FUNCTION_BLOCK Multicast_Client (* Basic Function Block Type *)
  (* Standard: 61499-2 *)
  (* Version 0.2, 2003-12-04, JHC, Rockwell Automation, Renamed for better indexing. *)
  (* Version 0.1, 2002-11-05, JHC, Rockwell Automation, Corrected missing ST element in Algorithm REQ. *)
  (* Version 0.0, 2000-05-30, JHC, Rockwell Automation *)
  (* Compiler header: package fb.rt.cs725; *)
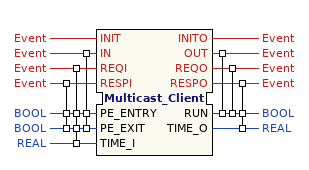
  EVENT_INPUT
    INIT; (* Initialization Request *)
    IN WITH PE_ENTRY, PE_EXIT;
    REQI WITH PE_ENTRY, PE_EXIT, TIME_I;
    RESPI WITH PE_ENTRY, PE_EXIT;
  END_EVENT
  EVENT_OUTPUT
    INITO; (* Initialization Confirm *)
    OUT WITH RUN;
    REQO WITH RUN;
    RESPO WITH RUN, TIME_O;
  END_EVENT
  VAR_INPUT
    PE_ENTRY : BOOL;
    PE_EXIT : BOOL;
    TIME_I : REAL;
  END_VAR
  VAR_OUTPUT
    RUN : BOOL;
    TIME_O : REAL;
  END_VAR
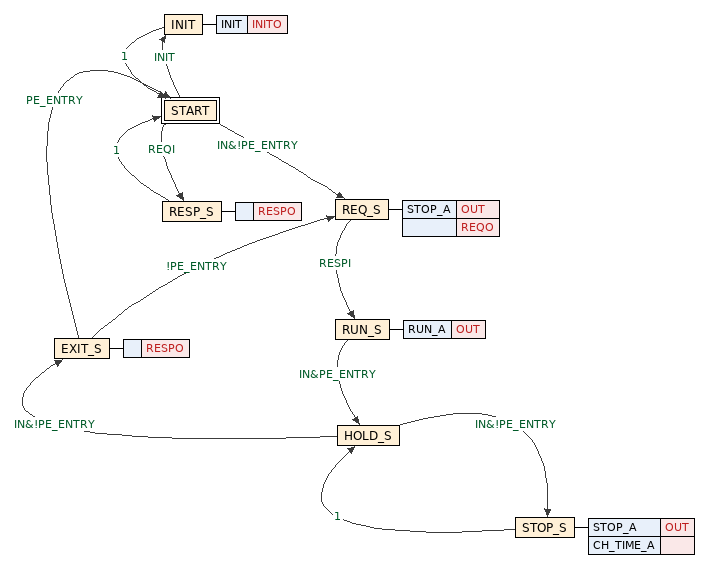
  EC_STATES
    START; (* Initial State *)
    INIT : INIT -> INITO; (* Initialization *)
    REQ_S : STOP_A -> OUT, -> REQO;
    RUN_S : RUN_A -> OUT;
    RESP_S : -> RESPO;
    EXIT_S : -> RESPO;
    STOP_S : STOP_A -> OUT, CH_TIME_A;
    HOLD_S;
  END_STATES
  EC_TRANSITIONS
    START TO INIT := INIT;
    INIT TO START := 1;
    START TO REQ_S := IN&!PE_ENTRY;
    REQ_S TO RUN_S := RESPI;
    START TO RESP_S := REQI;
    RESP_S TO START := 1;
    EXIT_S TO START := PE_ENTRY;
    RUN_S TO HOLD_S := IN&PE_ENTRY;
    HOLD_S TO EXIT_S := IN&!PE_ENTRY;
    HOLD_S TO STOP_S := IN&!PE_ENTRY;
    EXIT_S TO REQ_S := !PE_ENTRY;
    STOP_S TO HOLD_S := 1;
  END_TRANSITIONS
  ALGORITHM INIT IN Java: (* Initialization algorithm *)
RUN.value = true;
TIME_O.value = 0;
TIME_I.value = 0;
  END_ALGORITHM
  ALGORITHM RUN_A IN Java:
RUN.value = true;

System.out.println("RUNNING A");
  END_ALGORITHM
  ALGORITHM STOP_A IN Java:
RUN.value = false;

System.out.println("STOPPING");
  END_ALGORITHM
  ALGORITHM CH_TIME_A IN Java:
//if (TIME_I.value < TIME_O.value) {
//RESPO.serviceEvent(this);
//}

System.out.println("STATUS TEST");
  END_ALGORITHM
  ALGORITHM UPD_TIME_A IN Java:
if (TIME_O.value < TIME_I.value) {
TIME_O.value = TIME_I.value + 1;
} else {
TIME_O.value += 1;
}
  END_ALGORITHM
END_FUNCTION_BLOCK
